// TwinCAT 3 PLC project eHub
// ProgramVersion: 3.1.4023.0
// libraries:
//   Tc2_Standard, * (Beckhoff Automation GmbH)
//   Tc2_System, * (Beckhoff Automation GmbH)
//   Tc2_Utilities, * (Beckhoff Automation GmbH)
//   Tc3_Module, * (Beckhoff Automation GmbH)
// project tree:
//   DUTs/ E_EncoderType.TcDUT, E_IoDevice_ConnectionType.TcDUT, E_LabelStatus.TcDUT, E_MultiLightMode.TcDUT, E_ScannerResult.TcDUT, E_ScannerStatus.TcDUT, E_ScannerType.TcDUT, ST_BufferStats.TcDUT, ST_EncAr.TcDUT, ST_Heartbeat.TcDUT, ST_HornLightAr.TcDUT, ST_IODevice.TcDUT, ST_Msg_Buffer.TcDUT, ST_MultiLightAr.TcDUT, ST_OutDepOutAr.TcDUT, ST_ScanAr.TcDUT, ST_SCP.TcDUT, ST_StaticOutput.TcDUT, ST_User.TcDUT
//   GVLs/ vConst.TcGVL, vCore.TcGVL, vMessages.TcGVL
//   / PlcTask.TcTTO
//   POUs/ MAIN.TcPOU, P800_Core_Messaging.TcPOU, sMsg_Add_Core_Heartbeat.TcPOU, sMsg_Add_Message.TcPOU, sMsg_Process_Buffer.TcPOU, sMsg_Process_Queue.TcPOU, sMsg_SCP_Error.TcPOU, sMsg_SCP_Event.TcPOU, sMsg_SCP_Event_Num.TcPOU
// real-time tasks:
//   TASK PlcTask: cycle T#10ms, priority 20, ADS port 350

CONFIGURATION eHub
    RESOURCE PLC ON TwinCAT3
        TASK PlcTask(INTERVAL := T#10ms, PRIORITY := 20);
        PROGRAM MAIN WITH PlcTask : MAIN;
    END_RESOURCE
END_CONFIGURATION

// ---- DUTs/E_EncoderType.TcDUT
{attribute 'qualified_only'}
{attribute 'strict'}
TYPE E_EncoderType :
(
    LETE            := 0,
	LELE            := 1,
	Quad            := 3,
	PEP             := 4,
	Timer           := 5,
	Inc				:= 6
);
END_TYPE

// ---- DUTs/E_IoDevice_ConnectionType.TcDUT
{attribute 'qualified_only'}
{attribute 'strict'}
TYPE E_IoDevice_ConnectionType :
(
    None := 0,              // the connection state is ignored (always FALSE)
	Strict := 1,            // the connection state can never vary 
    Timed := 2              // the connection is OFF if the timeout is violated
);
END_TYPE

// ---- DUTs/E_LabelStatus.TcDUT
//{attribute 'qualified_only'}
//{attribute 'strict'}
TYPE E_LabelStatus :
(
	Good 		:= 0,
	LoBoy 		:= 1,
	NoData		:= 2,
	DataError	:= 3
);
END_TYPE

// ---- DUTs/E_MultiLightMode.TcDUT
{attribute 'qualified_only'}
{attribute 'strict'}
TYPE E_MultiLightMode :
(
	Off := 0,
	Red := 1,
	Yel := 2,
	Grn := 3,
	Blu := 4,
	BlinkRed := 5,
	BlinkYel := 6,
	BlinkGrn := 7,
	BlinkBlu := 8,
	ChangeRedYel := 9,
	ChangeRedGrn := 10,
	ChangeRedBlu := 11,
	ChangeYelGrn := 12,
	ChangeYelBlu := 13,
	ChangeGrnBlu := 14,
	PulseRed := 15,
	PulseYel := 16,
	PulseGrn := 17 
);
END_TYPE

// ---- DUTs/E_ScannerResult.TcDUT
{attribute 'qualified_only'}
{attribute 'strict'}
TYPE E_ScannerResult :
(
	None := 0,
	GoodRead := 1,
	NoRead := 2,
	LabelConflict := 3,
	NoData := 4,
	Overflow := 5 
);
END_TYPE

// ---- DUTs/E_ScannerStatus.TcDUT
{attribute 'qualified_only'}
{attribute 'strict'}
TYPE E_ScannerStatus :
(
	Offline := 0,
	Online := 1,
	Ready := 2,
	Busy := 3,
	Faulted := 4
);
END_TYPE

// ---- DUTs/E_ScannerType.TcDUT
{attribute 'qualified_only'}
{attribute 'strict'}
TYPE E_ScannerType :
(
	RS232			:= 1,		// RS232 Port on an I/O station
	GigE			:= 3,		// Gig-E camera
	AxiomEIP		:= 4,		// Axiom scanner with EIP connection
	SickEIP			:= 5,		// Sick scanner with a EIP
	Anybus			:= 8,		// Scanner with an Anybus converter
	SickEipCan		:= 10,		// Sick scanner with a EIP/Canbus connection
	DataLogic		:= 11,		// DataLogix scanner with EIP connection
	Turk			:= 12,		// Scanner connected to a Turck I/O station
	CognexHard		:= 13,		// Cognex with EIP, hardware triggered by sensor
	PhxGW			:= 14,		// Phoenix Contact ASCII-EIP Gateway
	CognexSoft		:= 15,		// Cognex with EIP trigger
	CognexInSight	:= 16,		// Cognex with EIP trigger
	UDP				:= 17,		// UDP socket
    Cognex90Buffer	:= 18,		// Cognex with EIP trigger - single buffer v90 update
	TcpClient		:= 19,		// TCP client
	PhxRsSlice		:= 21,		// Phoenix Contact Green RS232 or RS-485/422 slice
	BeckRsSlice		:= 22,		// Beckhoff EL6001 RS-232 or EL6021 RS-422/485 slice
	Sim				:= 99		// used for simulations
);
END_TYPE

// ---- DUTs/ST_BufferStats.TcDUT
TYPE ST_BufferStats :
STRUCT
	RDYcnt : DINT;
	ACKcnt : DINT;
	WatchdofTimeoutCnt	:DINT;
END_STRUCT
END_TYPE

// ---- DUTs/ST_EncAr.TcDUT
TYPE ST_EncAr :
STRUCT
    Tic                     :BOOL;
	
    Typ                     :E_EncoderType;
    
	ChA                     :INT;		// Channel A
    ChB                     :INT;
    ChC                     :INT;
    ChD                     :INT;
    ChE                     :INT;

    LastSignal              :BYTE;      // used by quad encoders to track the last channel that signalled
	LowByte					:UINT;      //analog input for incremental
	HighByte				:UINT;		//analog input for incremental
	Pos						:UINT;		//position
	LPos					:UINT;		//last scan position
	LFPos					:UINT;		//last forward position
	Change					:INT;		//change of current scan cycle
	LChange					:UINT;		//change of last scan
	Rotation				:UINT;		//change from last Z input (ChE)
	LRotation				:UINT;		//change of last full rotation
	Backwards				:BOOL;		//previous motion was backwards
	BackRollover			:USINT;		//number of times motion has rolled over backwards
	FaultDetectActivate     :INT;       // input that when latched activates the fault detect logic (typically a motor aux)
	FaultTimeout            :UDINT;		// if a tic does not occure within this timeout (x100ms) the encoder is flagged as faulted, max change for Incremental type
    FaultTmr                :UDINT;
	Fault_Reset				:INT;       // DI that resets the fault status
    IsFaulted               :BOOL;
	Rollover				:UINT;		// highest value the inc encoder can have before rolling over
	
	Motor					:INT;		// optional add-on for Timer type encoders. A tic will not be generated unless the motor is running.
	
	TicsPerSec				:UDINT;		// a count of the number of tics per second
	TicsPerSecAcc			:UDINT;
	FPMRatio				:REAL;		// a configured number needed to calculate the FPM
	FPM						:UINT;		// calculated feet per minute
	
	PPI						:REAL;		// encoder pulses per inch. Optional.

	IoConnIdx               :INT;       // the index into the IoDeviceAr so we can see if the encoder is connected
END_STRUCT
END_TYPE

// ---- DUTs/ST_Heartbeat.TcDUT
TYPE ST_Heartbeat :
STRUCT
	RespTmr 				:UDINT;         // how long DB took to respond (xScans)
	ReqTmr		    		:UINT;          // how long the request is hanging out there (xScans) 
	PollInterval			:UINT := 500;   // heartbeat polling interval (xScans)
	LastRespTime			:UDINT;         // scan time for last message handshake (xScans)
	Disabled 				:BOOL := FALSE;
	HostAck					:BOOL;          // host sets this to 1 = heartbeat
	HeartAttackCounter 		:UDINT;
	StressTestTarget		:UDINT;
END_STRUCT
END_TYPE

// ---- DUTs/ST_HornLightAr.TcDUT
TYPE ST_HornLightAr :
STRUCT
    Output      :UINT;
    On          :BOOL;
END_STRUCT
END_TYPE

// ---- DUTs/ST_IODevice.TcDUT
TYPE ST_IODevice :
STRUCT
	DevID			:INT;
	Typ				:E_IoDevice_ConnectionType;
	Connected		:BOOL;		    // TRUE = Connected
    StatusPt		:UINT;		    // analog input index for device state value
    StatusBit       :UINT := 999;   // bit of the StatusPt to check. 999 if evaluating the whole StatusPt	
	Status			:UINT;          // current status
	PrevStatus		:UINT;          // status on the previous scan cycle
    Timeout         :INT;           // for the "Timed" type, what is the timeout
	TimeoutTmr      :INT;           // used internally for timing
    
	GoodVal			:UINT;		    // the value when the device is connected
END_STRUCT
END_TYPE

// ---- DUTs/ST_Msg_Buffer.TcDUT
TYPE ST_Msg_Buffer :
STRUCT
    Pending         :STRING(4000);
    Sending         :STRING(4000);
    
    Ready           :BOOL;
    Ack             :BOOL;
	//ADSPubThrottle			:BOOL := TRUE;
	
	OverflowCount	:UINT;
    Stats			:ST_BufferStats;
    WatchDogTmr     :INT;      // toggles the Ready bit in case OPC/ADS falls asleep on the job
	
END_STRUCT
END_TYPE

// ---- DUTs/ST_MultiLightAr.TcDUT
TYPE ST_MultiLightAr :
STRUCT
	Red				:UINT;
	Yel				:UINT;
	Grn				:UINT;
	Blu				:UINT;
	Rate			:UINT;
	
	Mode			:E_MultiLightMode;
	Timer			:USINT;
	ColorInProc		:BOOL;
END_STRUCT
END_TYPE

// ---- DUTs/ST_OutDepOutAr.TcDUT
TYPE ST_OutDepOutAr :
STRUCT
    State                       :BOOL := 0;
    TestOutput                  :UINT := 0;         // output to monitor
    Output                      :UINT := 0;         // output to control
    OnDelay                     :UDINT := 0;        // configured on delay
    OffDelay                    :UDINT := 0;        // configured off delay

    OnCnt                       :UDINT := 0;        // how long the test output has been on
    OffCnt                      :UDINT := 0;        // how long the test output has been off
END_STRUCT
END_TYPE

// ---- DUTs/ST_ScanAr.TcDUT
TYPE ST_ScanAr :
STRUCT        
	Delimiter			:INT;
	ETX					:INT;
	STX					:INT;	
	NoReadChar			:INT;
	ConflictChar		:INT;
    IP					:STRING;	
	OverflowLmt			:INT;	
	Port				:INT;	
	MaxLength			:INT;
	Char1In				:INT;
	Char1Out			:INT;
	CxnState			:INT;
	Fault				:INT;
	SeqIn				:INT;
	SeqOut				:INT;
	LengthIn			:INT;
	LengthOut			:INT;
	TriggerOut			:INT;
	Setting				:ARRAY[1..15] OF DINT;	
	Typ					:E_ScannerType;
	TypInst				:INT;
	
	Status				:E_ScannerStatus;
	Result				:E_ScannerResult;
	Purge				:BOOL;					// set to clear the scanner of all data
	Busy				:BOOL;					// high on initial trigger, low when new sequence number arrives
	Error				:BYTE;
	HasLabels			:BOOL;
    Label1				:STRING(450);
	Label2				:STRING;
	Label3				:STRING;
	Label4				:STRING;
	Label5				:STRING;
	Label6				:STRING;	
	LabelIn				:USINT;
	LabelStatus			:E_LabelStatus;
	NoLabelCnt			:INT;	
	OverflowCnt			:INT;
	PrevLabel           :STRING;
	PrevBuffer     		:ARRAY[1..CORE_MAXSCANNER_BUFFERLEN] OF BYTE;		
	Trigger				:BOOL;					// set high when scanner isn't busy to initiate a scan	
	
	TxBuffer			:STRING(250);
END_STRUCT
END_TYPE

// ---- DUTs/ST_SCP.TcDUT
TYPE ST_SCP :
STRUCT
    IsConfigured          	:BOOL := FALSE;
	//IsCfgOK               :BOOL := FALSE;
	Init1stScan           	:BOOL;

    IORemoveAllForces     	:BOOL := FALSE;

	ScanCount             	:DINT;		// how many scan cycles have occured since startup
	ScanCountRollover     	:DINT;		// how many times ScanCount has rolled over (99 days 10:05:34)

	Tmr100msOscFlagLE     	:BOOL;
	Tmr100msOscFlag       	:BOOL;
	Tmr1sOscFlagLE        	:BOOL;
	Tmr1sOscFlag          	:BOOL;
	Rando				  	:DRAND;

	LogicActiveOut        	:UINT;		// output that turns ON when the logic is running
	FaultOut              	:UINT;		// output that turns ON if Error > 0

	Error                 	:UDINT;		// Error bits
	ErrorPrev             	:UDINT;		// Error bits
	ErrorAck              	:BOOL;		// resets the Error variable
	
    DisableMessaging      	:BOOL := FALSE;
	Heartbeat				:ST_Heartbeat;	//Heartbeat for SCP Buffer
	
	LinkLoss_ADS2DB			:BOOL := FALSE;
	LinkLoss_DB2ADS			:BOOL := FALSE;
	
	IsLicensed				:BOOL := FALSE;
END_STRUCT
END_TYPE

// ---- DUTs/ST_StaticOutput.TcDUT
TYPE ST_StaticOutput :
STRUCT
    Output          :INT;
    State           :BYTE;
END_STRUCT
END_TYPE

// ---- DUTs/ST_User.TcDUT
TYPE ST_User :
STRUCT
	MaskStart		:STRING;
	MaskEnd			:STRING;
	Timeout			:INT := 3000;
	
	Enabled			:BOOL;
	LoginState		:INT;
	LoginUser		:STRING;
	LoginRdy		:BOOL;
		
	User			:STRING;
	GoodUser		:BOOL;
	Tmr				:INT;
	LightCycle		:INT;
	LightTmr		:INT;
END_STRUCT
END_TYPE

// ---- GVLs/vConst.TcGVL
//
// This is an IOBuilder generated file
//
//      --- DO NOT EDIT OR OTHERWISE MODIFY THIS FILE ---
//
// Any future re-build will wipe out custom changes!
// If needed, create a new GVL or modify the PLCConstants table.
//
{attribute 'global_init_slot' := '40001'}
VAR_GLOBAL CONSTANT
	CB_MAXCARPLC                      :SINT := 1;
    CONV_MAXAXIS                      :INT := 1;       
    CONV_MAXBODICOPS                  :INT := 1;       
    CONV_MAXCTRLSTATIONS              :INT := 10;      
    CONV_MAXEMS                       :INT := 1;       // vConv.EmsAr[1..CONV_MAXMOTORS] OF ST_EMS
    CONV_MAXEMSINPUTS                 :INT := 6;       
	CONV_MAXSLUGDETECT       		  :INT := 50;
    CONV_MAXFLOWCTRL                  :INT := 50;      
    CONV_MAXGAPPERANALOG              :INT := 1;       // vConv.GapAnalog[1..CONV_MAXGAPPERANALOG] OF FB_Gapper_Analog
    CONV_MAXGAPPERPRESYNC             :INT := 1;       // vConv.GapPreSync[1..CONV_MAXGAPPERPRESYNC] OF FB_Gapper_PreSync
    CONV_MAXGAPPERQUE                 :INT := 20;      // Max number of cartons to track per gapper sync lane.
    CONV_MAXGAPPERS                   :INT := 5;       
    CONV_MAXIDXSLUGS                  :INT := 6;       
    CONV_MAXINVERTERS                 :INT := 100;     
    CONV_MAXJAMS                      :INT := 100;     
    CONV_MAXJAMZONES                  :INT := 20;      
    CONV_MAXMOTORDEPOUT               :INT := 1;       
    CONV_MAXMOTORDEPS                 :INT := 1;       // vConv.MotorDepAr[1..CONV_MAXMOTORDEPS] OF ST_MotorDepAr
    CONV_MAXMOTORS                    :INT := 100;     
    CONV_MAXOILERS                    :INT := 5;       
    CONV_MAXORPHANS                   :INT := 80;      
    CONV_MAXSYSINFEEDS                :INT := 1;       
    CONV_MAXTRAFFICCOP                :INT := 1;       
    CONV_MAXZONEHORNS                 :INT := 5;       
    CONV_MAXZONELIGHTS                :INT := 10;      
    CONV_MAXZONES                     :INT := 6;       
    CORE_MAXANALOGINPUTS              :INT := 100;     
    CORE_MAXANALOGOUTPUTS             :INT := 100;     
    CORE_MAXDEPOUTPUTS                :INT := 20;      
    CORE_MAXDIGITALINPUTS             :INT := 1000;    
    CORE_MAXDIGITALOUTPUTS            :INT := 1000;    
    CORE_MAXENCODERS                  :INT := 20;      
    CORE_MAXHORNS                     :INT := 20;      
    CORE_MAXLCAR                      :INT := 12;      // :ARRAY[0..CORE_MAXLCAR] OF ST_LightCurtain
    CORE_MAXLCI_EL6021                :INT := 4;       // :ARRAY[0..CORE_MAXLCI_EL6021] OF FB_BannerLightCurtain_EL6021_Quad
    CORE_MAXLIGHTS                    :INT := 20;      
    CORE_MAXMULTILIGHTS               :INT := 1;       // vCore.MultiLightAr[0..CORE_MAXMULTILIGHTS] OF ST_MultiLightAr
    CORE_MAXPLCDEVICES                :INT := 1;       // vCore.IODeviceAr[1..CORE_MAXPLCDEVICES] OF ST_IODevice
    CORE_MAXSCANNER_BUFFERLEN         :INT := 450;     
    CORE_MAXSCANNERS                  :INT := 32;      
    CORE_MAXSCANNERS_COGNEX           :INT := 1;       
    CORE_MAXSCANNERS_COGNEXINSIGHT    :INT := 1;       
    CORE_MAXSCANNERS_COGNEXSOFT       :INT := 1;       
    CORE_MAXSCANNERS_DATALOGIC        :INT := 1;       
    CORE_MAXSCANNERS_PHXGW            :INT := 1;
	CORE_MAXSCANNERS_PHXRSSLICE		  :INT := 1;
	CORE_MAXSCANNERS_BECKRSSLICE	  :INT := 1;
    CORE_MAXSCANNERS_SICK             :INT := 1;       
    CORE_MAXSCANNERS_SIM              :INT := 1;       
    CORE_MAXSCANNERS_UDP              :INT := 1;
	CORE_MAXSCANNERS_TCPCLIENT        :INT := 1;
    CORE_MAXSTATICOUTPUTS             :INT := 1;
    CORE_MAXSIMLABELS                 :INT := 1;       
    CTN_MAXALTLANES                   :INT := 10;      
    CTN_MAXASSIGNSLOTS                :INT := 300;     
    CTN_MAXCARTONAR                   :INT := 3000;    // Max number of cartons that can be tracked across all sorters.
    CTN_MAXDEVDIVERT                  :INT := 1;       // vCtn.Dev_Divert[1..CTN_MAXDEVDIVERT]
    CTN_MAXDEVEND                     :INT := 1;       
    CTN_MAXDEVENDDIV                  :INT := 1;       
    CTN_MAXDEVICECARTONS              :INT := 500;     // vCtn.Device[].CartonList[CTN_MAXDEVICECARTONS]
    CTN_MAXDEVICES                    :INT := 50;      
    CTN_MAXDEVLETETRK                 :INT := 1;       // vCtn.Dev_LETETracking[1..CTN_MAXDEVLETETRK]
    CTN_MAXDEVMDR2REG                 :INT := 1;       
    CTN_MAXDEVRCVSCAN                 :INT := 1;       
    CTN_MAXDEVSCALE                   :INT := 1;       
    CTN_MAXDEVSCANNER                 :INT := 2;       
    CTN_MAXDEVSFSTART                 :INT := 1;       
    CTN_MAXDEVSFSWIN                  :INT := 1;       
    CTN_MAXDEVSFSWOUT                 :INT := 1;       
    CTN_MAXDEVSHOEINDUCT              :INT := 1;       
    CTN_MAXDEVTRACKING                :INT := 1;       
    CTN_MAXLANES                      :INT := 20;      
    CTN_MAXSHOEDIVERTERS              :INT := 20;      
    CTN_MAXSHOES                      :INT := 3000;    // Number of Shoes tracked on a shoe sorter. Arbitrary. Change in BluePaw (vConst.CTN_MAXSHOES) if y
    CTN_MAXSORTERS                    :INT := 4;
	IDX0                              :INT := 0;
	IDX1                              :INT := 1;
	IDX2                              :INT := 2;
	IDX3                              :INT := 3;
	IDX4                              :INT := 4;
	IDX5                              :INT := 5;
    IND_MAX_TRA                       :INT := 1;       // FB_DI_Instance.TRA_*_Ar[0..IND_MAXDIPKG]
    IND_MAXDIINSTANCES                :INT := 1;       // vInd.DI[0..IND_MAXDIINSTANCES]
    IND_MAXDIPKG                      :INT := 10;      // FB_DI_Instance.PKGAr[0..IND_MAXDIPKG]
    IND_MAXDIZAR                      :INT := 1;       // vInd.DIZ[0..IND_MAXDIINSTANCES, 0..IND_MAXDIZAR]
    IND_MAXLKDAR                      :INT := 1;       // vInd.LKDAr[0..IND_MAXDIINSTANCES, 0..IND_MAXLKDAR]
    IND_MAXWIDPC                      :INT := 15;      // FB_DI_Instance.WID_PC_LOC_Ar[0..IND_MAXWIDPC]
    ITM_MAXCSORTCHUTES                :INT := 1200;    
    ITM_MAXDROPS                      :INT := 1;       // vItm.DropAr[1....ITM_MAXDROPS] OF ST_Itm_DropAr
    ITM_MAXITEMDETECTPES              :INT := 10;      
    ITM_MAXJAMBITSCLRDLIST            :INT := 32;      
    ITM_MAXJAMZONES                   :INT := 20;      
    ITM_MAXTUNEALIGNIDX1              :INT := 2000;    
    ITM_MAXTUNEALIGNIDX2              :INT := 200;     
    MDR_MAXBEDS                       :INT := 2000;    
    MDR_MAXINBOUNDCTNS                :INT := 10;      // vMDR.Bed[].Cartons[1..MDR_MAXINBOUNDCTNS]
    MDR_MAXLANEMAPS                   :INT := 10;      // Max lane mappings to a divert direction. See vMDR.Bed[].Lanes[1..3, MDR_MAXLANEMAPS]
    MDR_MAXMERGES                     :INT := 1;       
    MDR_MAXSLAVEDFWDOUTPUTS           :INT := 10;      // vMDR.Bed[].SlavedFwdOutputs[1..MDR_MAXSLAVEDFWDOUTPUTS]
    MRG_MAXCOMBINER                   :INT := 1;       // vConv.CombinerMerge[1..MRG_MAXCOMBINER]
    MRG_MAXINFEEDS                    :INT := 10;      
    MRG_MAXMDRINFEEDS                 :INT := 2;       
    MRG_MAXMDRMERGES                  :INT := 1;       
    MRG_MAXMERGES                     :INT := 6;       
    MRG_MAXRACETRACKS                 :INT := 6;       
    MRG_MAXZIPPER                     :INT := 1;       // vConv.ZipperMerge[1..MRG_MAXZIPPER]
    MRG_MAXZIPPERSLOTS                :INT := 1000;    
    SF_MAXBLOCKVAL                    :INT := 1;       
    SF_MAXEMPTY                       :INT := 1;       
    SF_MAXEMPTYSWIN                   :INT := 1;       
    SF_MAXINDUCT                      :INT := 1;       
    SF_MAXPACK                        :INT := 1;       
    SF_MAXSEP                         :INT := 1;       
    SF_MAXSLUGGER                     :INT := 6;       
    SF_MAXSWIN                        :INT := 1;       
    SF_MAXSWINSLUG                    :INT := 500;     
	SF_MAXUSW						  :INT := 1;
	SF_MAXUASSIGNSLOTS				  :INT := 1000;  
	PA_MAXPRINTER					  :INT := 1;					  
END_VAR

// ---- GVLs/vCore.TcGVL
//{attribute 'qualified_only'}
VAR_GLOBAL

    SCP                                 :ST_SCP;
    
	i									:INT;
    j									:DINT;
	
	// Input processing
    InputAr                             :ARRAY[0..CORE_MAXDIGITALINPUTS] OF UINT;	// this must start at [0]
	InputAr_DebOn						:ARRAY[0..CORE_MAXDIGITALINPUTS] OF INT;	// this must start at [0]
	InputAr_DebOff						:ARRAY[0..CORE_MAXDIGITALINPUTS] OF INT;	// this must start at [0]
	InputAr_GlitchLimit					:ARRAY[0..CORE_MAXDIGITALINPUTS] OF INT;	// this must start at [0]
    //InputAr_Config                      :ARRAY[1..CORE_MAXDIGITALINPUTS] OF ST_InputAr_Config;
	
    InputAr_RemoveAllForces             :BOOL := 0;	
    InputAr_Count                       :INT;
	InputRuntimeAr						:ARRAY[0..CORE_MAXDIGITALINPUTS] OF UINT;
    AInputAr                            :ARRAY[0..CORE_MAXANALOGINPUTS] OF UDINT;

    FindInput                           :BOOL;
    FindInputAr                         :ARRAY[1..10] OF UINT;
    FindInput_ptr                       :INT;

	ForcesIn							:ARRAY[0..MaxForceCollection] OF INT;
	ForcesOut							:ARRAY[0..MaxForceCollection] OF INT;
	ForcesMotor							:ARRAY[0..MaxForceCollection] OF INT;
	
	IODeviceAr							:ARRAY[0..CORE_MAXPLCDEVICES] OF ST_IODevice;
	IODevice_Count						:INT;
	
    // Scope
    //Scope								:ST_ScopeAr;
    
    // Output processing
    OutputAr                            :ARRAY[0..CORE_MAXDIGITALOUTPUTS] OF UINT;	// this must start at [0]
    OutputAr_RemoveAllForces            :BOOL := 0;
    OutputAr_Count                      :INT;
	OutputRuntimeAr                     :ARRAY[0..CORE_MAXDIGITALOUTPUTS] OF UINT;
    AOutputAr                           :ARRAY[0..CORE_MAXANALOGOUTPUTS] OF UDINT;
    StaticOutputAr                      :ARRAY[0..CORE_MAXSTATICOUTPUTS] OF ST_StaticOutput;
    StaticOutputAr_Count                :INT;
    
	HornAr_Count                        :UINT;
	HornAr                              :ARRAY[0..CORE_MAXHORNS] OF ST_HornLightAr;
	LightAr_Count                       :UINT;
	LightAr                             :ARRAY[0..CORE_MAXLIGHTS] OF ST_HornLightAr;
	MultiLightAr_Count					:UINT;
	MultiLightAr						:ARRAY[0..CORE_MAXMULTILIGHTS] OF ST_MultiLightAr;	
    OutDepAr_Count                      :UINT;
    OutDepAr                            :ARRAY[0..CORE_MAXDEPOUTPUTS] OF ST_OutDepOutAr;
	EncAr_Count                         :UINT;
    EncAr                               :ARRAY[0..CORE_MAXENCODERS] OF ST_EncAr;
	
	ScanAr_Count                        :INT;
    ScanAr                              :ARRAY[0..CORE_MAXSCANNERS] OF ST_ScanAr;
	ScanAr_ManualPurge					:ARRAY[0..CORE_MAXSCANNERS] OF BOOL;


	StationUser							:ARRAY[0..13] OF ST_User;
	
END_VAR


VAR_GLOBAL CONSTANT

	InBit_LE                    :INT := 0;
	InBit_Present               :INT := 1;
	InBit_Latch                 :INT := 2;
	InBit_TE                    :INT := 3;
    InBit_DetectState           :INT := 4;
    InBit_ForceState            :INT := 5;
    InBit_Forced                :INT := 6;	

   	OutBit_State                :INT := 0;    
	OutBit_Voltage              :INT := 1;
    OutBit_OnIsLow              :INT := 2;
    OutBit_Forced               :INT := 3;
    OutBit_ForceState           :INT := 4;

	ScanError_WriteFailure		:INT := 0;
	ScanError_ReadFailure 		:INT := 1;
	ScanError_DeviceFailure 	:INT := 2;
	ScanError_Timeout 			:INT := 3;
	ScanError_BadData 			:INT := 4;
	ScanError_LabelSize			:INT := 5;			// The size of a label is larger than a Label field can hold. Increase the label buffer size.
	ScanLabel_NoDest			:STRING := '0';
	ScanLabel_Overflow			:STRING := '-';
    
	ErrBit_Overflow				:INT := 0;			// one of the msg buffers has overflowed
	ErrBit_Heartbeat			:INT := 1;
	ErrBit_NoCtnSlots			:INT := 2;			// ctn.Carton[] slots are all being used
	ErrBit_ArrayViolation		:INT := 3;			// array bounds violation in the configuration
	ErrBit_LinkLoss_DB2ADS		:INT := 4;			// DB2ADS Service has lost connectivity to database
	ErrBit_LinkLoss_ADS2DB		:INT := 5;			// ADS2DB Service has lost connectivity to database
	ErrBit_NoJams				:INT := 6;			// no jams defined. we should at least have an e-stop as a jam so a "no-jam" configuration is not valid. 
	
	MaxForceCollection			:INT := 100;
END_VAR

// ---- GVLs/vMessages.TcGVL
//{attribute 'qualified_only'}
VAR_GLOBAL
    Msgs_SCP                :ST_Msg_Buffer;
    Msgs_Itm                :ST_Msg_Buffer;
    Msgs_Ind				:ST_Msg_Buffer;
	Msgs_Log				:ST_Msg_Buffer;
	Msgs_Stat				:ST_Msg_Buffer;
    
    Msgs_Test_Num           :UINT;
    
    //------------------------------------------------------------------------------------------------------------------------
    // Client Custom    10,000+
	//MsgCode_Some_Client_Specific_Message			:DINT := 10001;
	
    //------------------------------------------------------------------------------------------------------------------------
    // SCP level messages   0 - 49
    MsgCode_SCP_Event                               :DINT := 1;
    MsgCode_SCP_Heartbeat                           :DINT := 2;
    MsgCode_SCP_Error                               :DINT := 4;
    MsgCode_SCP_NeedConfig                          :DINT := 11;

    MsgCode_IO_Scope                                :DINT := 20;
	
    //------------------------------------------------------------------------------------------------------------------------
    // SCP level events   200 - 299
    Evt_SCP_BadConfig_Trk							:DINT := 201;
	Evt_SCP_BadConfig_Zone							:DINT := 202;
	Evt_SCP_BadConfig_Mrg							:DINT := 203;
	Evt_SCP_BadConfig_Gap							:DINT := 204;
	Evt_SCP_BadConfig_MDR							:DINT := 205;
	Evt_SCP_BadConfig_Scan							:DINT := 206;
	Evt_SCP_BadConfig_LightBar						:DINT := 224;
	Evt_SCP_BadConfig_Scale							:DINT := 219;
	Evt_SCP_Heartbeat_StressTest					:DINT := 214; //There are other events defined in the EventDef table between 206-213
	Evt_SCP_IsConfigured							:DINT := 216;
    Evt_SCP_DeviceConnected                      	:DINT := 217;
    Evt_SCP_DeviceDisconnected						:DINT := 218;

    //------------------------------------------------------------------------------------------------------------------------
    // Core component events   400 - 499
	Evt_Core_EncoderFailure        					:DINT := 401;
	Evt_IO_Glitch			      					:DINT := 402;
	Evt_Core_EncoderIncFwdRollJmpBck				:DINT := 403;
	Evt_Core_EncoderIncFwdJumpFwd					:DINT := 404;
	Evt_Core_EncoderIncFwdRollXJmpZero				:DINT := 405;
	Evt_Core_EncoderIncFwdRollJmpFwd				:DINT := 406;
	Evt_Core_EncoderIncFwdXJmpZero					:DINT := 407;
	Evt_Core_EncoderIncFwdJmpBck					:DINT := 408;
	Evt_Core_EncoderIncBckJmpFwd					:DINT := 409;
	Evt_Core_EncoderIncBckRollXJmpFwd				:DINT := 410;
	Evt_Core_EncoderIncBckRollJmpFwd				:DINT := 411;
	Evt_Core_EncoderIncBckXJmpZero					:DINT := 412;
	Evt_Core_EncoderIncBckJmpBck					:DINT := 413;

	Evt_Core_TcpSocket_Connected					:DINT := 420;
	Evt_Core_TcpSocket_ConnFailed					:DINT := 421;
	Evt_Core_TcpSocket_Closed						:DINT := 422;
	Evt_Core_TcpSocket_SendFailed					:DINT := 423;
	Evt_Core_TcpSocket_ReceiveFailed				:DINT := 424;
	Evt_Core_TcpSocket_CloseError					:DINT := 425;
	Evt_Core_TcpSocket_BufferFull					:DINT := 426;
	
	
	//------------------------------------------------------------------------------------------------------------------------
    // Conveyor Messages        = 50-99
    MsgCode_Conv_ZoneStart                          :DINT := 50;
    MsgCode_Conv_ZoneStop                           :DINT := 51;
    MsgCode_Conv_ZoneJammed                         :DINT := 52;
    MsgCode_Conv_JamStatus                          :DINT := 53;
	MsgCode_Conv_ZipperMerge_Alignment				:DINT := 60;	
    //------------------------------------------------------------------------------------------------------------------------
    // Conveyor Events        = 50-99
	Evt_Conv_SlugParams								:DINT := 220;
	
    //------------------------------------------------------------------------------------------------------------------------
    // CtnSort messages (200-299)
	MsgCode_Ctn_SorterError							:DINT := 200;
    MsgCode_Ctn_DestReq            					:DINT := 201;
	MsgCode_Ctn_Weight             					:DINT := 202;
    MsgCode_Ctn_Confirm            					:DINT := 203;
    MsgCode_Ctn_Recirc             					:DINT := 204;
    MsgCode_Ctn_LaneStatus         					:DINT := 205;
    MsgCode_Ctn_RcvScan            					:DINT := 206;
	MsgCode_Ctn_Alignment          					:DINT := 210;
    MsgCode_Ctn_PhasePerShoe       					:DINT := 211;
    MsgCode_Ctn_ShoeDivertOffset   					:DINT := 212;
    MsgCode_Ctn_GetSimLabels       					:DINT := 213;
    MsgCode_Ctn_TrackingError      					:DINT := 214;
    //------------------------------------------------------------------------------------------------------------------------
    // CtnSort events (2000-2999)
	//Codes currently same last 3 digits as v5.5, KU 7/20/18
	Evt_Ctn_WeightNoLabel         					:DINT := 2004;
	Evt_Ctn_WeightOverflow        					:DINT := 2005;
	Evt_Ctn_RcvScanFailed         					:DINT := 2007;
	Evt_Ctn_SorterStarted         					:DINT := 2008;
	Evt_Ctn_SorterStopped         					:DINT := 2009;
	Evt_Ctn_HostDestRedirect      					:DINT := 2010;
	Evt_Ctn_CartonTooLong         					:DINT := 2011;
	Evt_Ctn_InvalidAssignLost     					:DINT := 2012;
	Evt_Ctn_InvalidAssignLane     					:DINT := 2013;
	Evt_Ctn_InvalidAssignSeq      					:DINT := 2014;
	Evt_Ctn_LateCartonAssign      					:DINT := 2015;
	Evt_Ctn_UnexpectedCarton      					:DINT := 2016;
	Evt_Ctn_TrackingErrLate       					:DINT := 2017;
	Evt_Ctn_TrackingWarLate       					:DINT := 2018;
	Evt_Ctn_TrackingErrEarly      					:DINT := 2019;
	Evt_Ctn_TrackingWarEarly      					:DINT := 2020;
	Evt_Ctn_MissingShoeDetect     					:DINT := 2021;
	Evt_Ctn_ScannerOverflow       					:DINT := 2022;
	Evt_Ctn_ScannerNoLabel        					:DINT := 2023;
	Evt_Ctn_ScannerInvNewCarton   					:DINT := 2024;
	Evt_Ctn_ScannerError							:DINT := 2025;


    
    //------------------------------------------------------------------------------------------------------------------------
    // itmSort Messages     400 - 499
    MsgCode_itm_Event           					:DINT := 401;
    MsgCode_itm_Batch_Induct    					:DINT := 402;
    MsgCode_itm_Divert          					:DINT := 403;
    MsgCode_itm_Confirm         					:DINT := 404;
    MsgCode_itm_Misfire         					:DINT := 405;
    MsgCode_itm_RedButton       					:DINT := 406;
    MsgCode_itm_SOF_Induct      					:DINT := 407;
    MsgCode_itm_Heartbeat       					:DINT := 408;
    MsgCode_itm_RecordStepPulse 					:DINT := 409;
    MsgCode_itm_UnexOpen        					:DINT := 410;
    MsgCode_itm_CalcCarrier1A   					:DINT := 411;
    MsgCode_itm_SorterJam       					:DINT := 412;
    MsgCode_itm_SeqNumFail      					:DINT := 413; // NEED TO TEST - as of 1/25/18
    MsgCode_itm_IndStats        					:DINT := 414; 
    MsgCode_itm_MisStats        					:DINT := 415; 
	MsgCode_Itm_ZoneStats 							:DINT := 416; 
	MsgCode_itm_CallCarrier							:DINT := 417;
	MsgCode_itm_SortrakMotor						:DINT := 419;
	MsgCode_itm_LabelMerge							:DINT := 420;
	MsgCode_itm_KeyedInduction						:DINT := 421;
	MsgCode_itm_DrivePPM							:DINT := 422;
	MsgCode_itm_LLAIM_IND							:DINT := 423;
	MsgCode_itm_LLAIM_DIV							:DINT := 424;
	MsgCode_itm_LLAIM_CNF							:DINT := 425;
	MsgCode_itm_LLAIM_MIS							:DINT := 426;
	MsgCode_itm_Recirc         						:DINT := 427;
	MsgCode_itm_ChuteStatus    						:DINT := 428;
	MsgCode_itm_BadgeScan      						:DINT := 429;
	MsgCode_itm_Start        						:DINT := 430;
	MsgCode_itm_Stop        						:DINT := 431;
	MsgCode_itm_CalcJams							:DINT := 434; //Used to send the updated OnDelay for ITM Jams

    // Set up the ItmSort Event Codes
	// -----------------------------------------------------------------------------
    EvtCode_Itm_InductShift1 						:DINT := 4001;
    EvtCode_Itm_InductShift2 						:DINT := 4002;
    EvtCode_Itm_ZoneShift1 							:DINT := 4003;
    EvtCode_Itm_ZoneShift2 							:DINT := 4004;
    EvtCode_Itm_MisfireShift1 						:DINT := 4005;
    EvtCode_Itm_MisfireShift2 						:DINT := 4006;
    EvtCode_Itm_InductCarrier 						:DINT := 4007;
    EvtCode_Itm_ZoneCarrier 						:DINT := 4008;
    EvtCode_Itm_MisfireCarrier 						:DINT := 4009;
    EvtCode_Itm_StepPulse 							:DINT := 4010;
    EvtCode_Itm_UnknownItem 						:DINT := 4011;
    EvtCode_Itm_DeadTray 							:DINT := 4012;
    EvtCode_Itm_LateAssign 							:DINT := 4013;
    EvtCode_Itm_InvalidLI 							:DINT := 4014;
	EvtCode_Itm_HalfOpenLI							:DINT := 4015;
	EvtCode_Itm_HBStressTest						:DINT := 4016;
	EvtCode_Itm_WksLocShift1 						:DINT := 4017;
    EvtCode_Itm_WksLocShift2 						:DINT := 4018;
	EvtCode_Itm_DriveStop	 						:DINT := 4019;
    EvtCode_Itm_CB_CarTimeout	 					:DINT := 4030;
	EvtCode_Itm_CB_NetOverrun 						:DINT := 4031;
	EvtCode_Itm_CB_Error 							:DINT := 4033;
	EvtCode_Itm_CB_DivFail							:DINT := 4034;
	EvtCode_Itm_CB_RecvFail							:DINT := 4035; 
	EvtCode_Itm_CB_ParamMsgSent						:DINT := 4036;
	EvtCode_Itm_CB_RunMsgSent						:DINT := 4037;
	EvtCode_Itm_CB_MsgReturn						:DINT := 4038;
	EvtCode_Itm_CB_Reconnect						:DINT := 4039;


    //------------------------------------------------------------------------------------------------------------------------
    // PandA Messages   nnnn-zzzz
	MsgCode_PA_DestReq								:DINT := 281;
	MsgCode_PA_Print								:DINT := 282;
	MsgCode_PA_PrinterStatus						:DINT := 283;
	MsgCode_PA_SfSepScan							:UINT := 284;
	MsgCode_PA_LateAssign							:DINT := 285;
	MsgCode_PA_Apply								:DINT := 286;
	MsgCode_PA_AssignResult							:DINT := 287;
	
    //------------------------------------------------------------------------------------------------------------------------
    // PandA events (2000-2999)    
	Evt_PA_SfSepRespRecv							:UINT := 2840;
	Evt_PandAApplicatorLow							:UINT := 2850;	//change this	
	
    //------------------------------------------------------------------------------------------------------------------------
    // MDR Messages     nnnn-zzzz
    
    MsgCode_Mdr_DestReq								:UINT := 301;
    MsgCode_Mdr_Confirm								:UINT := 302;
    MsgCode_Mdr_Recirc								:UINT := 303;
    MsgCode_Mdr_Tote_Scan							:UINT := 311;
    MsgCode_Mdr_Tote_ScanError						:UINT := 312;
    MsgCode_Mdr_Tote_Removed						:UINT := 313;
        

    //------------------------------------------------------------------------------------------------------------------------
    // SkyFall Messages     nnnn-zzzz
    MsgCode_Sf_Destreq		       					:DINT := 501;
	MsgCode_Sf_Confirm		       					:DINT := 502;
	MsgCode_Sf_Recirc		       					:DINT := 503;	
    MsgCode_Sf_InductScan       					:DINT := 504;
    MsgCode_Sf_InductRel        					:DINT := 505;	
	MsgCode_Sf_SwInScan         					:DINT := 506;
	MsgCode_Sf_SwInRel          					:DINT := 507;
	MsgCode_Sf_SwInSlugRel							:DINT := 508;
	MsgCode_Sf_SwInSlugCmp							:DINT := 509;
    MsgCode_Sf_PackScan           					:DINT := 510;
    MsgCode_Sf_PackSep1Rel        					:DINT := 511;
    MsgCode_Sf_PackSep2Rel        					:DINT := 512;
    MsgCode_Sf_ServiceScan       					:DINT := 514;
	MsgCode_Sf_ServiceBtn       					:DINT := 515;
	MsgCode_Sf_InductReset       					:DINT := 516;
	MsgCode_Sf_InductCartonScan						:DINT := 517;
	MsgCode_Sf_SwitchingDiag         				:DINT := 520;
	MsgCode_Sf_USwScan         						:DINT := 521;
	MsgCode_Sf_InductUserLog       					:DINT := 524;
    //------------------------------------------------------------------------------------------------------------------------
    // SkyFall Events
	EvtCode_Sf_Ind_SepJam         					:DINT := 5001;
	EvtCode_Sf_Ind_ScanTimeout         				:DINT := 5002;
	EvtCode_Sf_SwIn_ScanTimeout        				:DINT := 5100;
	EvtCode_Sf_SwIn_RescanNoShuttle    				:DINT := 5101;
	EvtCode_Sf_SwIn_Release	        				:DINT := 5102;	
	EvtCode_Sf_SwIn_Backwards        				:DINT := 5103;	
	EvtCode_Sf_SwIn_SlugEarlier1       				:DINT := 5104;
	EvtCode_Sf_SwIn_SlugEarlier2       				:DINT := 5105;
	EvtCode_Sf_SwIn_SlugPrev	       				:DINT := 5106;
	EvtCode_Sf_SwIn_SlugLater1       				:DINT := 5107;
	EvtCode_Sf_SwIn_SlugLater2       				:DINT := 5108;
	EvtCode_Sf_SwIn_SlugNotFound       				:DINT := 5109;	
	EvtCode_Sf_SwIn_SlugNoRead       				:DINT := 5110;
	EvtCode_Sf_SwIn_RelFail            				:DINT := 5111;
    EvtCode_Sf_SwIn_RelFailHold            			:DINT := 5112;	
	EvtCode_Sf_USw_DuplicateScan       				:DINT := 5160;	
	EvtCode_Sf_Pack_RescanNoShuttle       			:DINT := 5201;
	EvtCode_Sf_Pack_SepJam       					:DINT := 5202;
	EvtCode_Sf_Pack_ScanTimeout		       			:DINT := 5203;	
	EvtCode_Sf_BV_NewShuttle	       				:DINT := 5300;	
	EvtCode_Sf_BreakawayLog1       					:DINT := 5600;
	EvtCode_Sf_BreakawayLog2       					:DINT := 5601;
	EvtCode_Sf_BreakawayLog3       					:DINT := 5602;	
	EvtCode_Ferag_Skytrain_DriveFault       		:DINT := 5900;	
	EvtCode_Ferag_Skytrain_ServiceMode       		:DINT := 5901;	
	
	//------------------------------------------------------------------------------------------------------------------------
	// Stat Messages    601-700
	MsgCode_Stat_MotorUpTime                        :DINT := 601;
	MsgCode_Stat_ChuteHit                           :DINT := 602;   
	MsgCode_Stat_ChuteMisfire                       :DINT := 603;
	MsgCode_Stat_ChuteRecirc                        :DINT := 604;
	MsgCode_Stat_ChuteSuspend                       :DINT := 605;
	MsgCode_Stat_Jams                               :DINT := 606;
	MsgCode_Stat_OutputOnTime                       :DINT := 607;
	MsgCode_Stat_InputOnTime                        :DINT := 608;
	MsgCode_Stat_DivertStatus						:DINT := 609;
	
	
	
	// TripWire is used to prevent multiple services of a like type from connecting to the same plc
	// holds the host name of the service that is currently using it.
	// when a service first come online it will clear the string value then wait 1000ms and check that the string is still clear.
	// when the program is running it will write its host name into the value every time it interacts with the plc.
	// this way we can see who is currely using it.
	TripWire_DB2ADS         :STRING(256);
	TripWire_ADS2DB         :STRING(256);
	TripWire_ADS2WEB        :STRING(256);

	// used to count the number of SQL exceptions the services have.
	SQL_ExceptionFlag	:INT;
	SQL_ExceptionCount	:INT;
END_VAR

// ---- POUs/MAIN.TcPOU
PROGRAM MAIN
VAR
	nCounter			:INT := 1;
	sText				:STRING;
	bFlag				:BOOL;
	bQuit				:BOOL;
	
	step				:INT;
	nTimeout			:INT := 250;
END_VAR


IF bFlag THEN
	step := step + 1;
END_IF

IF step > nTimeout THEN
	//bFlag := FALSE;	// limit to 1 msg as a test
	
	sMsg_SCP_Event_Num(100,	nCounter, 0, 0, 0, 0, 0, 0);
	sMsg_SCP_Event_Num(100,	nCounter + 1, 0, 0, 0, 0, 0, 0);
	sMsg_SCP_Event_Num(100,	nCounter + 2, 0, 0, 0, 0, 0, 0);

	nCounter := nCounter + 3;
	IF nCounter > 32000 THEN nCounter := 1; END_IF

	step := 0;
END_IF




P800_Core_Messaging();

IF bQuit THEN
	bQuit := FALSE;
	vMessages.Msgs_SCP.Pending := 'quit';
END_IF

END_PROGRAM

// ---- POUs/sMsg_SCP_Event_Num.TcPOU
FUNCTION sMsg_SCP_Event_Num : INT
VAR_INPUT
	pEventCode			:DINT;
	pI1					:DINT;
	pI2					:DINT;
	pI3					:DINT;
	pI4					:DINT;
	pI5					:DINT;
	pI6					:DINT;
	pI7					:DINT;
END_VAR
VAR
END_VAR

sMsg_Add_Message(
    Msgs_SCP,                  			// Buffer to use
    9,                                  // Num Params
    MsgCode_SCP_Event, '',       		// message code
    pEventCode, '',						// event code
    pI1, '',	                       	// param 1 
    pI2, '',    	                   	// param 2
    pI3, '',                            // param 3
    pI4, '',                            // param 4
    pI5, '',                            // param 5
    pI6, '',                            // param 6
    pI7, '',                            // param 7
    0, '',                              // param 10
    0, '',                              // param 11
    0, '',                              // param 12
    0, '',                              // param 13
    0, '',                              // param 14
    0, '',                              // param 15
    0, '',                              // param 16
    0, '',                              // param 17
    0, '',                              // param 18
    0, '',                              // param 19
    0, '');                             // param 20

RETURN;

END_FUNCTION

// ---- POUs/sMsg_Add_Message.TcPOU
FUNCTION sMsg_Add_Message : BOOL
VAR_IN_OUT
    pBuffer             :ST_Msg_Buffer;
END_VAR
VAR_INPUT
    pNumParams          :UINT;		// the number of parameters to use, including the message code
    pIntParam01         :DINT;		// set to the Message Code
    pCharParam01        :STRING(450);        // default string length is 80 characters + 1 null termination character
    pIntParam02         :DINT;
    pCharParam02        :STRING(450);
    pIntParam03         :DINT;
    pCharParam03        :STRING(450);
    pIntParam04         :DINT;
    pCharParam04        :STRING(450);
    pIntParam05         :DINT;
    pCharParam05        :STRING(450);
    pIntParam06         :DINT;
    pCharParam06        :STRING(450);
    pIntParam07         :DINT;
    pCharParam07        :STRING(450);
    pIntParam08         :DINT;
    pCharParam08        :STRING(450);
    pIntParam09         :DINT;
    pCharParam09        :STRING(450);
    pIntParam10         :DINT;
    pCharParam10        :STRING(450);
    pIntParam11         :DINT;
    pCharParam11        :STRING(450);
    pIntParam12         :DINT;
    pCharParam12        :STRING(450);
    pIntParam13         :DINT;
    pCharParam13        :STRING(450);
    pIntParam14         :DINT;
    pCharParam14        :STRING(450);
    pIntParam15         :DINT;
    pCharParam15        :STRING(450);
    pIntParam16         :DINT;
    pCharParam16        :STRING(450);
    pIntParam17         :DINT;
    pCharParam17        :STRING(450);
    pIntParam18         :DINT;
    pCharParam18        :STRING(450);
    pIntParam19         :DINT;
    pCharParam19        :STRING(450);
    pIntParam20         :DINT;
    pCharParam20        :STRING(450);
END_VAR
VAR
    str       			:STRING(450);
    index     			:UDINT;
	temp_buff			:STRING(4000);
	msg_len				:UDINT;
	free_space			:UDINT;
END_VAR

Msgs_Test_Num := Msgs_Test_Num + 1;

// make sure there is something to do
IF pNumParams < 1 OR SCP.DisableMessaging THEN
    RETURN;
END_IF

// clear the temp buffer
memset(ADR(temp_buff), 0, SIZEOF(temp_buff));

// add a leading "<"
concat2(ADR(temp_buff), ADR('<'), ADR(temp_buff), SIZEOF(temp_buff));

// add the parameters
IF pCharParam01[0] > 0 THEN
	concat2(ADR(temp_buff), ADR(pCharParam01), ADR(temp_buff), SIZEOF(temp_buff));
ELSE
    str := DINT_TO_STRING(pIntParam01);
	concat2(ADR(temp_buff), ADR(str), ADR(temp_buff), SIZEOF(temp_buff));
END_IF;

IF pNumParams >= 2 THEN
	concat2(ADR(temp_buff), ADR(','), ADR(temp_buff), SIZEOF(temp_buff));
	IF pCharParam02[0] > 0 THEN
		str := pCharParam02;
	ELSE
    	str := DINT_TO_STRING(pIntParam02);
	END_IF;
	concat2(ADR(temp_buff), ADR(str), ADR(temp_buff), SIZEOF(temp_buff));
END_IF

IF pNumParams >= 3 THEN
	concat2(ADR(temp_buff), ADR(','), ADR(temp_buff), SIZEOF(temp_buff));
	IF pCharParam03[0] > 0 THEN
		str := pCharParam03;
	ELSE
    	str := DINT_TO_STRING(pIntParam03);
	END_IF
	concat2(ADR(temp_buff), ADR(str), ADR(temp_buff), SIZEOF(temp_buff));
END_IF

IF pNumParams >= 4 THEN
	concat2(ADR(temp_buff), ADR(','), ADR(temp_buff), SIZEOF(temp_buff));
	IF pCharParam04[0] > 0 THEN
		str := pCharParam04;
	ELSE
    	str := DINT_TO_STRING(pIntParam04);
	END_IF
	concat2(ADR(temp_buff), ADR(str), ADR(temp_buff), SIZEOF(temp_buff));
END_IF

IF pNumParams >= 5 THEN
	concat2(ADR(temp_buff), ADR(','), ADR(temp_buff), SIZEOF(temp_buff));
	IF pCharParam05[0] > 0 THEN
		str := pCharParam05;
	ELSE
    	str := DINT_TO_STRING(pIntParam05);
	END_IF
	concat2(ADR(temp_buff), ADR(str), ADR(temp_buff), SIZEOF(temp_buff));
END_IF

IF pNumParams >= 6 THEN
	concat2(ADR(temp_buff), ADR(','), ADR(temp_buff), SIZEOF(temp_buff));
	IF pCharParam06[0] > 0 THEN
		str := pCharParam06;
	ELSE
    	str := DINT_TO_STRING(pIntParam06);
	END_IF
	concat2(ADR(temp_buff), ADR(str), ADR(temp_buff), SIZEOF(temp_buff));
END_IF

IF pNumParams >= 7 THEN
	concat2(ADR(temp_buff), ADR(','), ADR(temp_buff), SIZEOF(temp_buff));
	IF pCharParam07[0] > 0 THEN
		str := pCharParam07;
	ELSE
    	str := DINT_TO_STRING(pIntParam07);
	END_IF
	concat2(ADR(temp_buff), ADR(str), ADR(temp_buff), SIZEOF(temp_buff));
END_IF

IF pNumParams >= 8 THEN
	concat2(ADR(temp_buff), ADR(','), ADR(temp_buff), SIZEOF(temp_buff));
	IF pCharParam08[0] > 0 THEN
		str := pCharParam08;
	ELSE
    	str := DINT_TO_STRING(pIntParam08);
	END_IF
	concat2(ADR(temp_buff), ADR(str), ADR(temp_buff), SIZEOF(temp_buff));
END_IF

IF pNumParams >= 9 THEN
	concat2(ADR(temp_buff), ADR(','), ADR(temp_buff), SIZEOF(temp_buff));
	IF pCharParam09[0] > 0 THEN
		str := pCharParam09;
	ELSE
    	str := DINT_TO_STRING(pIntParam09);
	END_IF
	concat2(ADR(temp_buff), ADR(str), ADR(temp_buff), SIZEOF(temp_buff));
END_IF

IF pNumParams >= 10 THEN
	concat2(ADR(temp_buff), ADR(','), ADR(temp_buff), SIZEOF(temp_buff));
	IF pCharParam10[0] > 0 THEN
		str := pCharParam10;
	ELSE
    	str := DINT_TO_STRING(pIntParam10);
	END_IF
	concat2(ADR(temp_buff), ADR(str), ADR(temp_buff), SIZEOF(temp_buff));
END_IF

IF pNumParams >= 11 THEN
	concat2(ADR(temp_buff), ADR(','), ADR(temp_buff), SIZEOF(temp_buff));
	IF pCharParam11[0] > 0 THEN
		str := pCharParam11;
	ELSE
    	str := DINT_TO_STRING(pIntParam11);
	END_IF
	concat2(ADR(temp_buff), ADR(str), ADR(temp_buff), SIZEOF(temp_buff));
END_IF

IF pNumParams >= 12 THEN
	concat2(ADR(temp_buff), ADR(','), ADR(temp_buff), SIZEOF(temp_buff));
	IF pCharParam12[0] > 0 THEN
		str := pCharParam12;
	ELSE
    	str := DINT_TO_STRING(pIntParam12);
	END_IF
	concat2(ADR(temp_buff), ADR(str), ADR(temp_buff), SIZEOF(temp_buff));
END_IF

IF pNumParams >= 13 THEN
	concat2(ADR(temp_buff), ADR(','), ADR(temp_buff), SIZEOF(temp_buff));
	IF pCharParam13[0] > 0 THEN
		str := pCharParam13;
	ELSE
    	str := DINT_TO_STRING(pIntParam13);
	END_IF
	concat2(ADR(temp_buff), ADR(str), ADR(temp_buff), SIZEOF(temp_buff));
END_IF

IF pNumParams >= 14 THEN
	concat2(ADR(temp_buff), ADR(','), ADR(temp_buff), SIZEOF(temp_buff));
	IF pCharParam14[0] > 0 THEN
		str := pCharParam14;
	ELSE
    	str := DINT_TO_STRING(pIntParam14);
	END_IF
	concat2(ADR(temp_buff), ADR(str), ADR(temp_buff), SIZEOF(temp_buff));
END_IF

IF pNumParams >= 15 THEN
	concat2(ADR(temp_buff), ADR(','), ADR(temp_buff), SIZEOF(temp_buff));
	IF pCharParam15[0] > 0 THEN
		str := pCharParam15;
	ELSE
    	str := DINT_TO_STRING(pIntParam15);
	END_IF
	concat2(ADR(temp_buff), ADR(str), ADR(temp_buff), SIZEOF(temp_buff));
END_IF

IF pNumParams >= 16 THEN
	concat2(ADR(temp_buff), ADR(','), ADR(temp_buff), SIZEOF(temp_buff));
	IF pCharParam16[0] > 0 THEN
		str := pCharParam16;
	ELSE
    	str := DINT_TO_STRING(pIntParam16);
	END_IF
	concat2(ADR(temp_buff), ADR(str), ADR(temp_buff), SIZEOF(temp_buff));
END_IF

IF pNumParams >= 17 THEN
	concat2(ADR(temp_buff), ADR(','), ADR(temp_buff), SIZEOF(temp_buff));
	IF pCharParam17[0] > 0 THEN
		str := pCharParam17;
	ELSE
    	str := DINT_TO_STRING(pIntParam17);
	END_IF
	concat2(ADR(temp_buff), ADR(str), ADR(temp_buff), SIZEOF(temp_buff));
END_IF

IF pNumParams >= 18 THEN
	concat2(ADR(temp_buff), ADR(','), ADR(temp_buff), SIZEOF(temp_buff));
	IF pCharParam18[0] > 0 THEN
		str := pCharParam18;
	ELSE
    	str := DINT_TO_STRING(pIntParam18);
	END_IF
	concat2(ADR(temp_buff), ADR(str), ADR(temp_buff), SIZEOF(temp_buff));
END_IF

IF pNumParams >= 19 THEN
	concat2(ADR(temp_buff), ADR(','), ADR(temp_buff), SIZEOF(temp_buff));
	IF pCharParam19[0] > 0 THEN
		str := pCharParam19;
	ELSE
    	str := DINT_TO_STRING(pIntParam19);
	END_IF
	concat2(ADR(temp_buff), ADR(str), ADR(temp_buff), SIZEOF(temp_buff));
END_IF

IF pNumParams >= 20 THEN
	concat2(ADR(temp_buff), ADR(','), ADR(temp_buff), SIZEOF(temp_buff));
	IF pCharParam20[0] > 0 THEN
		str := pCharParam20;
	ELSE
    	str := DINT_TO_STRING(pIntParam20);
	END_IF
	concat2(ADR(temp_buff), ADR(str), ADR(temp_buff), SIZEOF(temp_buff));
END_IF

// add a trailing ">"
concat2(ADR(temp_buff), ADR('>'), ADR(temp_buff), SIZEOF(temp_buff));

// now make sure the new message will fit into whatever remaining space is in the pending buffer
msg_len := LEN2(ADR(temp_buff));
free_space := 4000 - LEN2(ADR(pBuffer.Pending));

IF msg_len < free_space THEN
	concat2(ADR(pBuffer.Pending), ADR(temp_buff), ADR(pBuffer.Pending), SIZEOF(pBuffer.Pending));
ELSE
	pBuffer.OverflowCount := pBuffer.OverflowCount + 1;
	SCP.Error.ErrBit_Overflow := 1;
END_IF

RETURN;

END_FUNCTION

// ---- POUs/P800_Core_Messaging.TcPOU
PROGRAM P800_Core_Messaging
VAR
END_VAR

// if flag goes high from service set it low and bump counter
IF (vMessages.SQL_ExceptionFlag > 0) THEN
	vMessages.SQL_ExceptionFlag :=0;
	vMessages.SQL_ExceptionCount := SQL_ExceptionCount + 1;	
	// cap exception count
	IF (vMessages.SQL_ExceptionCount > 10001 )THEN
		vMessages.SQL_ExceptionCount := 10001;
	END_IF	
END_IF


IF SCP.DisableMessaging THEN
	RETURN;
END_IF

// Process whatever buffers you want here
sMsg_Process_Buffer(Msgs_SCP);      // generic SCP message buffer
sMsg_Process_Buffer(Msgs_Itm);      // Itmsort SCP message buffer
sMsg_Process_Buffer(Msgs_Ind);      // Itmsort FAST SCP message buffer
sMsg_Process_Buffer(Msgs_Log);      // Multithreaded, used for silent messages/heartbeat

END_PROGRAM

// ---- POUs/sMsg_Process_Buffer.TcPOU
FUNCTION sMsg_Process_Buffer : BOOL
VAR_IN_OUT
    pBuffer   : ST_Msg_Buffer;
END_VAR
VAR
    ptr     :UDINT;
    len     :UDINT;
END_VAR

IF pBuffer.Ack THEN
    pBuffer.Ack := FALSE;
    pBuffer.Ready := FALSE;
    pBuffer.Sending[IDX0] := 0;    // effectively indicates the buffer is empty
    pBuffer.WatchDogTmr := 0;
	pBuffer.Stats.ACKcnt := pBuffer.Stats.ACKcnt + 1;
	IF (pBuffer.Stats.ACKcnt >= 2147483500) THEN
		pBuffer.Stats.ACKcnt := 1;
	END_IF
	
END_IF

// if there is something pending and the sending is empty...
IF pBuffer.Pending[IDX0] > 0 AND pBuffer.Sending[IDX0] = 0 THEN
    // ... transfer pending to sending
    ptr := 0;
    WHILE pBuffer.Pending[ptr] > 0 AND ptr < 4000 DO
        pBuffer.Sending[ptr] := pBuffer.Pending[ptr];
        pBuffer.Pending[ptr] := 0;      // erase as we go along
        ptr := ptr + 1;
	END_WHILE
    pBuffer.Sending[ptr] := 0;   // don't forget to zero terminate the string
    
	pBuffer.Stats.RDYcnt := pBuffer.Stats.RDYcnt + 1;
	IF (pBuffer.Stats.RDYcnt >= 2147483500) THEN
		pBuffer.Stats.RDYcnt := 1;
	END_IF
	pBuffer.Ready := TRUE;
    pBuffer.WatchDogTmr := 0;     // time how long it takes to pick up this msg
END_IF
//(* removing the watchdog per Mike Higleys request. He states that toggling the Ready bit messes with the services - mjm
// if the sending buffer is active with data... 
IF pBuffer.Sending[IDX0] > 0 THEN
    // time how long until it's picked up
    pBuffer.WatchDogTmr := pBuffer.WatchDogTmr + 1;
    // if not within the timeout...   (25 = 100ms)
    IF pBuffer.WatchDogTmr = 25 THEN
        // toggle the Ready bit OFF
        pBuffer.Ready := FALSE;
		pBuffer.Stats.WatchdofTimeoutCnt := pBuffer.Stats.WatchdofTimeoutCnt + 1;
	END_IF
    IF pBuffer.WatchDogTmr = 51 THEN
        pBuffer.Ready := TRUE;
        pBuffer.WatchDogTmr := 0;
	END_IF
END_IF
//*)

END_FUNCTION

// ---- POUs/sMsg_Add_Core_Heartbeat.TcPOU
FUNCTION sMsg_Add_Core_Heartbeat : BOOL
VAR_INPUT
	nRespTime					:UDINT;
END_VAR
VAR
END_VAR

sMsg_Add_Message(
    Msgs_Log,                  			// Buffer to use
    2,                                  // Num Params
    MsgCode_SCP_Heartbeat, '',       	// param 1
    nRespTime, '',					// param 2
    0, '',              // param 3 
    0, '',                       		// param 4
    0, '',                             	// param 5
    0, '',                              // param 6
    0, '',                              // param 7
    0, '',                              // param 8
    0, '',                              // param 9
    0, '',                              // param 10
    0, '',                              // param 11
    0, '',                              // param 12
    0, '',                              // param 13
    0, '',                              // param 14
    0, '',                              // param 15
    0, '',                              // param 16
    0, '',                              // param 17
    0, '',                              // param 18
    0, '',                              // param 19
    0, '');                             // param 20

RETURN;

END_FUNCTION

// ---- POUs/sMsg_Process_Queue.TcPOU
FUNCTION sMsg_Process_Queue : BOOL
VAR_IN_OUT
    pBuffer   : ST_Msg_Buffer;
END_VAR
VAR
    str       			:STRING;
    index     			:UDINT;
	temp_buff			:STRING(4000);
	msg_len				:UDINT;
	free_space			:UDINT;
END_VAR

free_space := 4000 - LEN2(ADR(pBuffer.Pending));

//When there is data to work with and more than 10% free space, spin.
WHILE (pBuffer.MsgQ.Queue.Position[IDX1].HasData) AND (free_space > 400) DO
	// now make sure the new message will fit into whatever remaining space is in the pending buffer
	msg_len := LEN2(ADR(pBuffer.MsgQ.Queue.Position[IDX1].BufferString));
	free_space := 4000 - LEN2(ADR(pBuffer.Pending));
	
	IF msg_len < free_space THEN
		
		concat2(ADR(pBuffer.Pending), ADR(pBuffer.MsgQ.Queue.Position[IDX1].BufferString), ADR(pBuffer.Pending), SIZEOF(pBuffer.Pending));
		
		//cycle the stack
		pBuffer.MsgQ.QueueWorker.ShiftPositionArray(1);
	ELSE
		free_space := 0;
	END_IF
END_WHILE

END_FUNCTION

// ---- POUs/sMsg_SCP_Error.TcPOU
FUNCTION sMsg_SCP_Error : BOOL
VAR_INPUT
	Errors			:UDINT;
END_VAR
VAR
END_VAR

sMsg_Add_Message(
    Msgs_SCP,                  			// Buffer to use
    2,                                  // Num Params
    MsgCode_SCP_Error, '',              // param 1
    Errors, '',                         // param 2
    0, '',                              // param 3 
    0, '',                              // param 4
    0, '',                              // param 5
    0, '',                              // param 6
    0, '',                              // param 7
    0, '',                              // param 8
    0, '',                              // param 9
    0, '',                              // param 10
    0, '',                              // param 11
    0, '',                              // param 12
    0, '',                              // param 13
    0, '',                              // param 14
    0, '',                              // param 15
    0, '',                              // param 16
    0, '',                              // param 17
    0, '',                              // param 18
    0, '',                              // param 19
    0, '');                             // param 20

RETURN;

END_FUNCTION

// ---- POUs/sMsg_SCP_Event.TcPOU
FUNCTION sMsg_SCP_Event : INT
VAR_INPUT
	pEventCode			:DINT;
	pI1					:DINT;
	pS1					:STRING;
	pI2					:DINT;
	pS2					:STRING;
	pI3					:DINT;
	pS3					:STRING;
	pI4					:DINT;
	pS4					:STRING;
	pI5					:DINT;
	pS5					:STRING;
	pI6					:DINT;
	pS6					:STRING;
	pI7					:DINT;
	pS7					:STRING;
END_VAR
VAR
END_VAR

sMsg_Add_Message(
    Msgs_SCP,                  			// Buffer to use
    9,                                  // Num Params
    MsgCode_SCP_Event, '',       		// message code
    pEventCode, '',						// event code
    pI1, pS1,                       	// param 1 
    pI2, pS2,                       	// param 2
    pI3, pS3,                           // param 3
    pI4, pS4,                           // param 4
    pI5, pS5,                           // param 5
    pI6, pS6,                           // param 6
    pI7, pS7,                           // param 7
    0, '',                              // param 10
    0, '',                              // param 11
    0, '',                              // param 12
    0, '',                              // param 13
    0, '',                              // param 14
    0, '',                              // param 15
    0, '',                              // param 16
    0, '',                              // param 17
    0, '',                              // param 18
    0, '',                              // param 19
    0, '');                             // param 20

RETURN;

END_FUNCTION
